(* IEC 61131-3 sources: MotionTestBenchMaster/Logical/00_AID/Libraries/Sidel_Libraries/Powertoys, 10 files *)

(* ---- Powertoys.typ ---- *)
(********************************************************************
 * COPYRIGHT -- Bernecker + Rainer
 ********************************************************************
 * Library: Powertoys
 * File: Powertoys.typ
 * Author: gibertinim
 * Created: March 27, 2014
 ********************************************************************
 * Data types of library Powertoys
 ********************************************************************)
(********************************                    CUSTOM LOGGER ENTRY                   ***********************************************************)

TYPE
	pwr_log_custom_entry : 	STRUCT  (*Custom logger entry string*)
		adr_string : UDINT; (*Address of the ascii string*)
		len : UDINT; (*Length of the binary memory data*)
		adr_mem : UDINT; (*Address to the binary memory data*)
		errorNum : UINT; (*Error number to write*)
		logLevel : USINT; (*Information level*)
	END_STRUCT;
END_TYPE

(*********************************                            HARDWARE LIST                          **************************************************************)

TYPE
	searchIO_info_typ : 	STRUCT  (*Hardware information list*)
		Path : STRING[80]; (*Station path*)
		ModelNumber : STRING[80]; (*Model number*)
		Name : STRING[80]; (*Hw name*)
		Serial : UDINT; (*Serial number*)
	END_STRUCT;
END_TYPE

(********************************                              AXIS INFORMATIONS                **************************************************************)

TYPE
	pwlInfo_typ : 	STRUCT  (*Powerlink node properties datatype*)
		number : USINT; (*Number of Powerlink Module*)
		path : STRING[80]; (*Path of Powerlink Module*)
		description : STRING[80]; (*Description of Powerlink Module*)
		name : STRING[80]; (*Name of Powerlink Module*)
		modelNumber : STRING[80]; (*Module number of powerlink *)
		present : BOOL; (*Enable blinking*)
	END_STRUCT;
END_TYPE

(* ---- CleanMgr.st ---- *)
(********************************************************************
 * COPYRIGHT --
 ********************************************************************
 * Library: Powertoys
 * File: CleanMgr.st
 * Author: Administrator
 * Created: January 09, 2015
 ********************************************************************
 * Implementation of library Powertoys
 ********************************************************************)

(* Clean old files from a folder *)
FUNCTION_BLOCK CleanMgr

	IF enable THEN
		(* Function block enabled *)
		CASE step OF

			0:
				busy 		:= TRUE;
				ready		:= FALSE;
				error 		:= FALSE;
				errorID 	:= ERR_FUB_BUSY;

				(* Getting the input parameters *)
				memset(ADR(dirInfoData), 0, SIZEOF(dirInfoData));
				memset(ADR(oldestFile), 0, SIZEOF(oldestFile));
				tRefresh.PT 		:= refreshTime;
				getDirInfo.pDevice	:= adrPath;
				getDirInfo.pPath	:= ADR('//');
				getLastFileName.pDevice := adrPath;
				getLastFileName.pPath := ADR('//');
				getLastFileName.option := fiFILE;
				getLastFileName.data_len := SIZEOF(dirInfoData);
				deleteFile.pDevice := adrPath;
				step := 1;

				IF (refreshTime <= T#10ms) OR (adrPath = 0) OR (nrElements = 0) THEN

					(* Refresh time too low, or path address = 0, or numer of elements invalid *)
					step 		:= 200;
					errorStep 	:= 0;
					error 		:= TRUE;
					errorID 	:= ERR_BUR_ILLPAR;

				END_IF;

			1:
				(* Waiting the refresh timer *)
				tRefresh.IN := TRUE;

				IF (adrPath <> getDirInfo.pDevice) THEN
					(* Incorrect path address *)
					step 		:= 200;
					errorStep 	:= 1;
					error 		:= TRUE;
					errorID 	:= ERR_BUR_ILLPAR;

				ELSIF tRefresh.Q THEN

					getDirInfo.enable := TRUE;
					IF (getDirInfo.status = ERR_FUB_BUSY) THEN
	 					step := 10;
					END_IF;

				END_IF;

			10:
				tRefresh.IN := FALSE;

				IF (adrPath <> getDirInfo.pDevice) THEN
					(* Incorrect path address *)
					step 		:= 200;
					errorStep 	:= 1;
					error 		:= TRUE;
					errorID 	:= ERR_BUR_ILLPAR;

				ELSIF (getDirInfo.status = ERR_OK) THEN
					fileFound := getDirInfo.filenum;
					step := 11;

				ELSIF (getDirInfo.status <> ERR_OK) AND (getDirInfo.status <> ERR_FUB_BUSY) THEN

					(* Error *)
					step 		:= 200;
					errorStep 	:= 10;
					error 		:= TRUE;
					errorID 	:= getDirInfo.status;
				END_IF;

			11:
				IF (getDirInfo.filenum > nrElements) THEN

					(* Proceeding with cleanup *)
					step := 20;
				ELSE
					step := 0;
				END_IF;
				getDirInfo.enable	:= FALSE;

			20:
				(* Clean up, finding the oldest file *)
				memset(ADR(dirInfoData), 0, SIZEOF(dirInfoData));
				memset(ADR(oldestFile), 0, SIZEOF(oldestFile));
				cnt := 0;
				getLastFileName.entry := cnt;
				getLastFileName.pData := ADR(oldestFile);
				IF (adrPath <> getLastFileName.pDevice) THEN
					(* Incorrect path address *)
					step 		:= 200;
					errorStep 	:= 20;
					error 		:= TRUE;
					errorID 	:= ERR_BUR_ILLPAR;
				ELSE
					getLastFileName.enable := TRUE;
					step := 21;
				END_IF

			21:
				IF (adrPath <> getLastFileName.pDevice) THEN
					(* Incorrect path address *)
					step 		:= 200;
					errorStep 	:= 21;
					error 		:= TRUE;
					errorID 	:= ERR_BUR_ILLPAR;

				ELSIF (getLastFileName.status = ERR_OK) THEN
					memset(ADR(dirInfoData), 0, SIZEOF(dirInfoData));
					getLastFileName.enable := FALSE;
					step := 22;

				ELSIF ((getLastFileName.status <> ERR_OK) AND (getLastFileName.status <> ERR_FUB_BUSY)) THEN
					(* Error *)
					step 		:= 200;
					errorStep 	:= 20;
					error 		:= TRUE;
					errorID 	:= getLastFileName.status;
				END_IF;

			22:

				getLastFileName.pData := ADR(dirInfoData);
				cnt := cnt + 1;
				getLastFileName.entry := cnt;

				IF (cnt < fileFound) THEN

					step := 23;

				ELSE
					(* search finished *)
					step := 30;
				END_IF;

			23:
				getLastFileName.enable := TRUE;
				IF (adrPath <> getLastFileName.pDevice) THEN
					(* Incorrect path address *)
					step 		:= 200;
					errorStep 	:= 23;
					error 		:= TRUE;
					errorID 	:= ERR_BUR_ILLPAR;

				ELSIF (getLastFileName.status = ERR_OK) THEN
					getLastFileName.enable := FALSE;
					step := 24;

				ELSIF ((getLastFileName.status <> ERR_OK) AND (getLastFileName.status <> ERR_FUB_BUSY) AND (getLastFileName.status <> ERR_FUB_ENABLE_FALSE)) THEN
					(* Error *)
					step 		:= 200;
					errorStep 	:= 22;
					error 		:= TRUE;
					errorID 	:= getLastFileName.status;
				END_IF;

			24:
				(* Checking the file timestamp *)
				IF (dirInfoData.Date < oldestFile.Date) THEN
					memcpy(ADR(oldestFile), ADR(dirInfoData), SIZEOF (oldestFile));

				END_IF;

				memset(ADR(dirInfoData),0,SIZEOF (dirInfoData));
				step := 22;

			30:
				(* Search finished, deleting the oldest file *)
				deleteFile.pName := ADR(oldestFile.Filename[0]);
				deleteFile.enable := TRUE;
				IF (adrPath <> deleteFile.pDevice) THEN
					(* Incorrect path address *)
					step 		:= 200;
					errorStep 	:= 30;
					error 		:= TRUE;
					errorID 	:= ERR_BUR_ILLPAR;
				ELSIF (deleteFile.status = ERR_OK) THEN
					deleteFile.enable := FALSE;
					IF (fileFound - 1 > nrElements) THEN
						getDirInfo.enable := TRUE;
						step := 10;
					ELSE
						step := 0;
					END_IF;

				ELSIF (deleteFile.status <> ERR_OK) AND (deleteFile.status <> ERR_FUB_ENABLE_FALSE) AND (deleteFile.status <> ERR_FUB_BUSY) THEN
					(* Error *)
					step 		:= 200;
					errorStep 	:= 30;
					error 		:= TRUE;
					errorID 	:= deleteFile.status;
				END_IF;

			200:
				(* Error state, resetting all the internal function block *)
				tRefresh.IN				:= FALSE;
				getDirInfo.enable		:= FALSE;
				getLastFileName.enable	:= FALSE;
				deleteFile.enable		:= FALSE;

		END_CASE;

	ELSE

		(* Function block disabled, resetting all the internal fubs *)
		busy 		:= FALSE;
		ready		:= FALSE;
		error 		:= TRUE;
		errorID 	:= ERR_FUB_ENABLE_FALSE;

		step 		:= 0;
		errorStep 	:= 0;
		cnt 		:= 0;
		tRefresh.IN				:= FALSE;
		getDirInfo.enable		:= FALSE;
		getLastFileName.enable	:= FALSE;
		deleteFile.enable		:= FALSE;
	END_IF;

	tRefresh();
	getDirInfo();
	getLastFileName();
	deleteFile();
END_FUNCTION_BLOCK

(* ---- CustomLogEntry.st ---- *)
(********************************************************************
 * COPYRIGHT -- Bernecker + Rainer
 ********************************************************************
 * Library: Powertoys
 * File: CustomLogEntry.st
 * Author: gibertinim
 * Created: March 27, 2014
 ********************************************************************
 * Implementation of library Powertoys
 ********************************************************************)

(* Write a custom entry into the specified logger *)
FUNCTION_BLOCK CustomLogEntry

	IF enable THEN

		pEntry ACCESS adrCustomEntry;

		CASE step OF

			0:	(*Check if Log exist*)
				LogInfo.Name	:= 'userlog';
				LogInfo.Execute	:= TRUE;
				errorID 		:= ERR_FUB_BUSY;
				busy			:= TRUE;
				error			:= FALSE;

				IF (LogInfo.StatusID = arEVENTLOG_ERR_LOGBOOK_NOT_FOUND) THEN
					step := 5;
					LogInfo.Execute	:= FALSE;
				ELSIF (LogInfo.Done AND LogInfo.StatusID = ERR_OK) THEN
					step 			:= 10;
					LogIdent		:= LogInfo.Ident;
					LogInfo.Execute	:= FALSE;
				END_IF

			5:	(*Create Log*)
				LogCreate.Name			:= 'userlog';
				LogCreate.Size			:= 4096;	//4096 BYTES
				LogCreate.Persistence	:= arEVENTLOG_PERSISTENCE_PERSIST;
				LogCreate.Execute		:= TRUE;
				errorID 				:= ERR_FUB_BUSY;
				busy					:= TRUE;
				error					:= FALSE;

				IF LogCreate.Error THEN
					step 		:= 200;
					error		:= TRUE;
					errorID		:= LogInfo.StatusID;
					errorStep	:= 1;
				ELSIF (LogCreate.Done AND LogInfo.StatusID = ERR_OK) THEN
					step				:= 10;
					LogIdent			:= LogCreate.Ident;
					LogCreate.Execute	:= FALSE;
				END_IF

			10:	(* Writing the logger informations  *)
				eventID := ArEventLogMakeEventID(
					Severity := pEntry.logLevel,
					Facility := 0,
					ErrorCode := pEntry.errorNum);

				LogWrite.EventID		:= eventID;
				LogWrite.Ident			:= LogIdent;
				LogWrite.AddData		:= pEntry.adr_string;
				LogWrite.AddDataSize	:= 80;
				LogWrite.AddDataFormat	:= 1;
				LogWrite.Execute		:= TRUE;

				(* Waiting until the log is written succesfully *)
				IF (LogWrite.Done AND LogWrite.StatusID = ERR_OK) THEN
					(* Log entry written succesfully*)
					step := 101;
					LogWrite.Execute := FALSE;
				ELSIF LogWrite.Error THEN
					(* Error occured while saving the logger *)
					errorStep	:= 10;
					errorID		:= LogWrite.StatusID;
					error		:= TRUE;
					step		:= 200;
				END_IF;

			101:
				done := TRUE;
				busy := FALSE;
				errorID := ERR_OK;

			200:
				(* Error step *)
				LogCreate.Execute	:= FALSE;
				LogWrite.Execute	:= FALSE;
				LogInfo.Execute		:= FALSE;
				done				:= TRUE;
				busy				:= FALSE;
		END_CASE;

	ELSE
		error				:= FALSE;
		errorID				:= ERR_FUB_ENABLE_FALSE;
		errorStep			:= 0;
		step	 			:= 0;
		LogCreate.Execute	:= FALSE;
		LogWrite.Execute	:= FALSE;
		LogInfo.Execute		:= FALSE;
		done				:= FALSE;
		busy				:= FALSE;

	END_IF;

	LogCreate();
	LogWrite();
	LogInfo();

END_FUNCTION_BLOCK

(* ---- PlkList.st ---- *)
(********************************************************************
 * COPYRIGHT --
 ********************************************************************
 * Library: Powertoys
 * File: Plk_list.st
 * Author: Administrator
 * Created: July 04, 2014
 ********************************************************************
 * Implementation of library Powertoys
 ********************************************************************)

(* Powerlink list *)
FUNCTION_BLOCK PlkList

	IF (enable	=	TRUE) THEN

		CASE step OF

			0: (* Choosing the operating mode
					0 = standard memory consumption
					1 = low memory consumption - slowest
				*)
				errorID 		:=	ERR_FUB_BUSY;
				busy			:=	TRUE;
				error			:=	FALSE;
				done			:= 	FALSE;

				IF (mode = 0) THEN
					step 		:= 1;
				ELSIF (mode = 1) THEN
					step 		:= 10;
				ELSE
					(* Wrong mode *)
					step		:= 200;
					error 		:= TRUE;
					errorID		:= ERR_NOTIMPLEMENTED;
					errorStep	:= 0;
					busy		:= FALSE;
					done		:= FALSE;
				END_IF;

			1:
				(* Getting the whole hardware list *)
				searchIO_0.adrSearchIO 	:= ADR(searchIoData);
				searchIO_0.mode 		:= asdiagALL;
				searchIO_0.wholeList	:= TRUE;
				searchIO_0.enable		:= TRUE;

				IF (searchIO_0.errorID = ERR_FUB_BUSY) THEN
					step := 2;
				END_IF;

			2:
				IF ((searchIO_0.errorID	=	ERR_OK) AND (searchIO_0.done = TRUE)) THEN

					(*resetting array and variables*)

					strcpy(ADR(tmpPlkInterface), ADR(plkInterface));
					strcat(ADR(tmpPlkInterface),ADR('.'));
					step		:=	3;
					indexInfo	:=	0;
					indexPwl	:=	0;

				ELSIF ((searchIO_0.errorID	<>	ERR_OK)	AND	(searchIO_0.errorID	<>	ERR_FUB_BUSY)) THEN

					(* Going to the error state *)
					errorID		:=	searchIO_0.errorID;
					errorStep	:=	1;
					step		:=	200;
					error		:=	TRUE;
				END_IF

			3: (*saving inside an array	(ArrayStringTemp) the path hardware longer than plk inteface*)
			IF (indexInfo	<	searchIO_0.nrEntries)	THEN

				(* Ci metto tutto quello dopo SS1.IF1
					Es:
					ST2
					ST3
					ST5.IF1

				*)
				IF 	strlen(ADR(searchIoData[indexInfo].Path))	>=	strlen(ADR(tmpPlkInterface))	THEN
					strcpy(ADR(ArrayStringTemp[indexPwl]),(ADR(searchIoData[indexInfo].Path)+ strlen(ADR(tmpPlkInterface))));
					arrayIndexPwl[indexPwl]	:=	indexInfo;
					indexPwl				:=	indexPwl+1;
				END_IF;

				indexInfo	:=	indexInfo+1;
			ELSE
				step		:=	4;
				oldIndexPwl :=	indexPwl;

				indexPwl	:=	0;

				indexInfo	:=	0;
				indexPwl2	:=	0;
				dotFound	:=	FALSE;

				END_IF;

		4:
			(*Finding dot or string null inside elements of temp array*)
			IF (indexPwl	<	strlen(ADR(ArrayStringTemp[indexInfo]))	OR	strlen(ADR(ArrayStringTemp[indexInfo]))	=	0 )	THEN

				IF (memcmp(ADR(ArrayStringTemp[indexInfo])+indexPwl,ADR('.'),1)	=0	)	THEN
					step		:=	5;
					indexPwl	:=	0;
					dotFound 	:= TRUE;
				END_IF;

			ELSE
				step		:=	5;
				indexPwl	:=	0;

			END_IF;
			indexPwl	:=	indexPwl+1;

		5:

			(*if there isn't a dot, the string is our node powerlink*)
			IF (dotFound	=	FALSE) THEN

				pData ACCESS (adrPlkInfo + indexPwl2*SIZEOF(pData));
				pData.number	:=	arrayIndexPwl[indexInfo];

				IF strlen(ADR(searchIoData[arrayIndexPwl[indexInfo]].ModelNumber))	<>	0 	AND
					pData.number	<>	0									THEN
					(* Powerlink node present *)
					pData.present	:=	TRUE;
				ELSE
					(* Powerlink node not present *)
					pData.present	:=	FALSE;
				END_IF;

				(*Copying information about powerlink node*)
				strcpy(ADR(pData.path),						ADR(ArrayStringTemp[indexInfo]));
				strcpy(ADR(pData.modelNumber),				ADR(searchIoData[arrayIndexPwl[indexInfo]].ModelNumber));
				strcpy(ADR(pData.name),						ADR(searchIoData[arrayIndexPwl[indexInfo]].Name));
				strcpy(ADR(ArrayStringTemp2[indexPwl2]),	ADR(ArrayStringTemp[indexInfo]));
				arrayIndexPwl2[indexPwl2]					:=	arrayIndexPwl[indexInfo];
				indexPwl2									:=	indexPwl2+1;

			END_IF;
			(**)
			indexInfo	:=	indexInfo+1;
			IF (indexInfo	<	oldIndexPwl) THEN

				dotFound	:=	FALSE;
				step	:=	4;

			ELSE

				step	:=	6;

			END_IF;

		6:
			busy := FALSE;
			done := TRUE;
			errorID := ERR_OK;

			entryFound := indexPwl2;

			10:
				(* Low memory consumption mode *)
				(* In this mode each entry is processe one by one instead of processing the whole list *)
				(* Getting the whole hardware list *)
				searchIO_0.adrSearchIO 	:= ADR(searchIoData);
				searchIO_0.mode 		:= asdiagALL;
				searchIO_0.wholeList	:= FALSE;
				searchIO_0.enable		:= TRUE;
				indexInfo 				:= 0;
				indexPwl2 				:= 0;
				(* Getting informations from the first hw found *)
				searchIO_0.stationIndex	:= 0;

				IF (searchIO_0.errorID = ERR_FUB_BUSY) THEN
					step := 11;
				END_IF;

			11:

				IF ((searchIO_0.errorID	=	ERR_OK) AND (searchIO_0.done = TRUE)) THEN

					(*resetting array and variables*)

					strcpy(ADR(tmpPlkInterface), ADR(plkInterface));
					strcat(ADR(tmpPlkInterface),ADR('.'));
					step		:=	12;
					nrIO 		:= searchIO_0.nrEntries;

				ELSIF ((searchIO_0.errorID	<>	ERR_OK)	AND	(searchIO_0.errorID	<>	ERR_FUB_BUSY)) THEN
					(* Going to the error state *)
					errorID		:=	searchIO_0.errorID;
					errorStep	:=	10;
					step		:=	200;
					error		:=	TRUE;
				END_IF

			12:
				 (* Se la lunghezza del path trovato dalla search io è maggiore o uguale a quello dell'interfaccia powerlink, allora è un probabile nodo powerlink *)
				(* Copio nella variabile temporanea solo quello che viene dopo i caratteri che compongono l'interfaccia powerlink:
				Es: Ci metto tutto quello dopo SS1.IF1

				in powerlink if ci deve finire 'SS1.IF1.'

				Se per esempio avremo come entry:
				SS1.IF1
				SS1.IF1.ST2
				SS1.IF1.ST3
				SSI.IF1.ST5.IF8

				RIMARRANNO

				ST2
				ST3
				ST5.IF8

				*)
				IF 	strlen(ADR(searchIoData[0].Path))	>=	strlen(ADR(tmpPlkInterface))	THEN

					(* Possible powerlink node *)
					strcpy(ADR(ArrayStringTemp[0]),(ADR(searchIoData[0].Path)+ strlen(ADR(tmpPlkInterface))));

					arrayIndexPwl[0]	:=	indexInfo;

					step := 13;

				ELSE
					(* Not a powerlink node *)
					step := 100;
				END_IF;

			13:
				(* If the remaining temporary string is empty, this is the powerlink inferface, not the powerlink node  *)

				IF (strlen(ADR(ArrayStringTemp[0])) <> 0) THEN

					(* Possible powerlink node *)
					tmpCnt		:= 0;
					step		:= 14;
				ELSE
					(* Not a powerlink node *)
					step		:= 100;
				END_IF;

			14:
				(* I have only something like:
				ST5
				ST41
				ST123
				ST41.IFblablabla
				ST12

				I can say that if there is not the dot, this is a powerlink node

				SEARCHING inside of the string if there is the dot
				*)
				IF (tmpCnt < strlen(ADR(ArrayStringTemp[0]))) THEN

					IF (memcmp(ADR(ArrayStringTemp[0])+tmpCnt,ADR('.'),1)	= 0	) THEN

						(* Dot found, this is not a powerlink node *)
						step := 100;

					ELSE
						tmpCnt := tmpCnt + 1;
					END_IF;

				ELSE
					(* This is a powerlink node *)
					step := 15;
				END_IF;

			15:
				(* Collecting data of the powerlink node *)
				pData ACCESS (adrPlkInfo + indexPwl2*SIZEOF(pData));
				pData.number	:=	indexInfo;

				IF strlen(ADR(searchIoData[0].ModelNumber))	<>	0 	AND
					pData.number	<>	0									THEN
					(* Powerlink node present *)
					pData.present	:=	TRUE;
				ELSE
					(* Powerlink node not present *)
					pData.present	:=	FALSE;
				END_IF;

				(*Copying information about powerlink node*)
				strcpy(ADR(pData.path),						ADR(ArrayStringTemp[0]));
				strcpy(ADR(pData.modelNumber),				ADR(searchIoData[0].ModelNumber));
				strcpy(ADR(pData.name),						ADR(searchIoData[0].Name));
				indexPwl2									:=	indexPwl2+1;

				step	:=	100;

			100:
				(* Not a powerlink node, processing a new entry *)
				searchIO_0.enable		:= FALSE;

				IF (searchIO_0.errorID = ERR_FUB_ENABLE_FALSE) THEN
					indexInfo := indexInfo + 1;
					step := 101;
				END_IF;

			101:
				(* Checking if I have to read an other entry *)
				IF ((indexInfo < nrIO)AND(indexPwl < nrEntry))  THEN

					(* Cleaning temporary variables *)
					memset(ADR(searchIoData),0,SIZEOF(searchIoData));

					(* Going to process a new entry *)
					step := 102;

				ELSE

					(* Sequence finished *)
					step := 120;

				END_IF;

			102:
				(* Reading a new search IO entry *)
				searchIO_0.adrSearchIO 	:= ADR(searchIoData);
				searchIO_0.mode 		:= asdiagALL;
				searchIO_0.wholeList	:= FALSE;
				searchIO_0.enable		:= TRUE;

				(* Getting informations from the first hw found *)
				searchIO_0.stationIndex	:= indexInfo;

				IF (searchIO_0.errorID = ERR_FUB_BUSY) THEN
					step := 103;
				END_IF;

			103:

				IF ((searchIO_0.errorID	=	ERR_OK) AND (searchIO_0.done = TRUE)) THEN

					(*resetting array and variables*)

					step		:=	12;
					nrIO 		:= searchIO_0.nrEntries;

				ELSIF ((searchIO_0.errorID	<>	ERR_OK)	AND	(searchIO_0.errorID	<>	ERR_FUB_BUSY)) THEN
					(* Going to the error state *)
					errorID		:=	searchIO_0.errorID;
					errorStep	:=	102;
					step		:=	200;
					error		:=	TRUE;
				END_IF

			120:
			(* Sequence completed *)
				done 				:= TRUE;
				busy 				:= FALSE;
				error 				:= FALSE;
				errorID				:= ERR_OK;
				searchIO_0.enable	:= FALSE;
				entryFound := indexPwl2;

			200:
				(* Error state, disabling all the used function block and waiting  for enable = false *)
				searchIO_0.enable 	:= FALSE;

		END_CASE;

	ELSE
		(* Function block not enabled *)
		error				:= TRUE;
		errorID				:= ERR_FUB_ENABLE_FALSE;

		(* Resetting  the internal variables *)
		errorStep			:= 0;
		step	 			:= 0;

		memset(ADR(arrayIndexPwl),		0,	SIZEOF(arrayIndexPwl));
		memset(ADR(ArrayStringTemp),	0,	SIZEOF(ArrayStringTemp));
		memset(ADR(arrayIndexPwl2),		0,	SIZEOF(arrayIndexPwl2));
		memset(ADR(ArrayStringTemp2),	0,	SIZEOF(ArrayStringTemp2));
		memset(ADR(tmpPlkInterface),	0,	SIZEOF(tmpPlkInterface));

		step		:=	0;
		indexInfo	:=	0;
		indexPwl	:=	0;
		indexPwl2	:=	0;
		entryFound 	:= 	0;
		nrIO		:=	0;
		done				:= FALSE;
		busy				:= FALSE;

		(* Disabling the block *)
		searchIO_0.enable 	:= FALSE;

	END_IF;

	(*Function Block Call*)
	searchIO_0();
END_FUNCTION_BLOCK

(* ---- Powertoys.fun ---- *)
(********************************************************************
 * COPYRIGHT -- Bernecker + Rainer
 ********************************************************************
 * Library: Powertoys
 * File: Powertoys.fun
 * Author: gibertinim
 * Created: March 27, 2014
 ********************************************************************
 * Functions and function blocks of library Powertoys
 ********************************************************************)

FUNCTION_BLOCK CustomLogEntry (*Write a custom entry into the specified logger*)
	VAR_INPUT
		enable : BOOL; (*Enable the function block*)
		adrCustomEntry : UDINT; (*Address of the custom entry*)
	END_VAR
	VAR_OUTPUT
		busy : BOOL; (*True when the function block is busy*)
		error : BOOL; (*True when the function block is in error*)
		errorID : DINT; (*Current error ID*)
		done : BOOL; (*True when the entry is succesfully written*)
	END_VAR
	VAR
		LogCreate : ArEventLogCreate;
		LogInfo : ArEventLogGetIdent; (*Get the information from the specified logger*)
		LogWrite : ArEventLogWrite; (*Write the entry into the logger*)
		eventID : DINT;
		errorStep : UINT; (*Internal error step*)
		pEntry : REFERENCE TO pwr_log_custom_entry; (*Pointer to the custom entry*)
		step : USINT; (*Internal fub step*)
		LogIdent : ArEventLogIdentType;
	END_VAR
END_FUNCTION_BLOCK

FUNCTION_BLOCK SearchIO (*Function Block to show hardware list component*)
	VAR_INPUT
		enable : BOOL; (*Enable the function block*)
		adrSearchIO : UDINT; (*Address of the search io data structure*)
		wholeList : BOOL; (*True to create the hw list, false for a single entries*)
		stationIndex : UDINT; (*Station index number (used only if wholeList = FALSE)*)
		mode : UDINT; (*Operating mode*)
	END_VAR
	VAR_OUTPUT
		busy : BOOL; (*True when the function block is busy*)
		done : BOOL; (*True when the data are ready*)
		error : BOOL; (*True when the function block is in error*)
		errorID : UINT; (*Current error ID*)
		nrEntries : UDINT; (*Number of entries found*)
	END_VAR
	VAR
		counter : UDINT; (*Internal counter*)
		ident : UDINT; (*Identifier*)
		FB_DiagGetStrInfo : DiagGetStrInfo; (*Get the string information of the module*)
		FB_DiagCreateInfo : DiagCreateInfo; (*Collect the information of the specified module*)
		FB_DiagGetNumInfo : DiagGetNumInfo; (*Get the numeric information from the specified module*)
		step : USINT; (*Internal fub step*)
		errorStep : USINT; (*Internal error step*)
		pData : REFERENCE TO searchIO_info_typ; (*Pointer to the data structure*)
	END_VAR
END_FUNCTION_BLOCK

FUNCTION_BLOCK PlkList (*Powerlink list*)
	VAR_INPUT
		enable : BOOL; (*Enable the function block*)
		adrPlkInfo : UDINT; (*Address of the powerlink information list*)
		mode : USINT; (*Fub operating mode (0 high memory usage, 1 low memory usage)*)
		nrEntry : UDINT; (*Number of powerlink elements to write on the list*)
		plkInterface : STRING[80]; (*String initialize a lenght of powerlink path*)
	END_VAR
	VAR_OUTPUT
		done : BOOL; (*Powerlink list complete*)
		busy : BOOL; (*Function block busy*)
		error : BOOL; (*Function block in error*)
		errorID : UINT; (*Function block error ID*)
		entryFound : USINT; (*Number of powerlink node in the configuration*)
	END_VAR
	VAR
		errorStep : USINT; (*Internal error step*)
		step : USINT; (*Internal step*)
		pData : REFERENCE TO pwlInfo_typ; (*Pointer to the powerlink list*)
		searchIO_0 : SearchIO; (*Search IO informations*)
		searchIoData : ARRAY[0..253] OF searchIO_info_typ; (*Search IO informations strusture*)
		arrayIndexPwl : ARRAY[0..253] OF USINT; (*Array to save index of hardware list complete*)
		arrayIndexPwl2 : ARRAY[0..253] OF USINT; (*Array to save index when dot is not finding*)
		ArrayStringTemp : ARRAY[0..253] OF STRING[80]; (*Array temp for saving name of powerlink node longer than plkinterface*)
		ArrayStringTemp2 : ARRAY[0..253] OF STRING[80]; (*Array to save path name when dot is not finding*)
		indexInfo : USINT; (*Index of number entries of harware list complete*)
		tmpPlkInterface : STRING[80]; (*Internal powerlink interface name*)
		indexPwl : USINT; (*Index of array for saving name of powerlink node longer than plkinterface*)
		oldIndexPwl : USINT; (*savind old index powerlink*)
		indexPwl2 : USINT; (*Index of array when dot is not finding*)
		dotFound : BOOL; (*Finding dot inside an array*)
		nrIO : UDINT; (*Number of IO found with the SEARCH IO fub*)
		tmpCnt : USINT; (*Temporary counter*)
	END_VAR
END_FUNCTION_BLOCK

FUNCTION_BLOCK profiMan (*Profiler archive manager*)
	VAR_INPUT
		enable : BOOL; (*Enable the function block*)
		refreshTime : TIME; (*Automatic refresh time*)
		maxArchive : USINT; (*Maximum number of profiler acrhive stored*)
		archiveListADR : UDINT; (*Address of the archive list*)
	END_VAR
	VAR_OUTPUT
		errorID : UINT; (*Current error ID*)
		valid : BOOL; (*True when the output data are valid*)
		error : BOOL; (*True when the function block is in error*)
		profilerStatus : USINT; (*Profiler status*)
		archiveFound : UDINT; (*Number of profiler archive found*)
		busy : BOOL; (*True when the function block is busy*)
		profStateActive : BOOL; (*Profiler active. AR profiler is ready.*)
		profStateStopped : BOOL; (*Data recording stopped.*)
		profStateRunning : BOOL; (*Data being recorded.*)
		profStateReady : BOOL; (*Data recording completed. The data module is ready to be evaluated (AS profiler).*)
		profStateR2R : BOOL; (*Ready to start. A profiling definition was installed successfully and can be started.*)
		profStateInactive : BOOL; (*Profiler inactive. Profiling cannot be carried out (AR profiler disabled in Sysconf).*)
		profStateR2Rman : BOOL; (*Ready to start (startup install). The profiler definition was installed successfully with the profMODE_NOAUTOSTART mode and can be started.*)
	END_VAR
	VAR
		pArchiveList : REFERENCE TO PROFILER_MODINFO; (*Pointer to the archive list*)
		step : USINT; (*Internal state machine step*)
		getProfStatus : LogStateGet; (*Get the status of the profiler*)
		errorStep : USINT; (*Internal error step*)
		getProfArchInfo : LogArchInfo; (*Gets profiler's archive informations*)
		refresh : TON; (*Refresh timer*)
	END_VAR
END_FUNCTION_BLOCK

FUNCTION_BLOCK sdmMAN (*Sdm configuration manager*)
	VAR_INPUT
		enable : BOOL; (*Enable the function block*)
		mode : USINT; (*Function block operating mode: 0 - SDM on, 1 - SDM off, 2 SDM status manual*)
		reqSDMstatus : UDINT; (*Requested SDM status*)
		pDumpDevice : UDINT; (*Pointer to the file device of the system dump*)
	END_VAR
	VAR_OUTPUT
		sdmStatus : UDINT; (*Actual SDM status*)
		busy : BOOL; (*True when the function block is working*)
		ready : BOOL; (*True when the function block is waiting for a change of reqSDMstatus*)
		error : BOOL; (*True when the function block is in error*)
		errorID : UINT; (*Actual error ID*)
		internalError : BOOL; (*Internal error*)
		errorStep : USINT; (*Actual error step*)
	END_VAR
	VAR
		old_mode : USINT; (*Old mode*)
		setSDMstatus : CfgSetSdmStatus; (*Set the sdm status*)
		getSDMstatus : CfgGetSdmStatus; (*Get the sdm status*)
		oldSdmStatus : UDINT; (*Old SDM status*)
		step : USINT; (*Internal function block step*)
		writeLogFlag : BOOL; (*Write an entry into the logger*)
		errorStepString : STRING[80]; (*Error step as string*)
		errorString : STRING[80]; (*Error string*)
		errorEntry : pwr_log_custom_entry; (*Log entry*)
		sDump : SdmSystemDump; (*Makes the system dump*)
		writeError : CustomLogEntry; (*Write the error into the user logger*)
	END_VAR
END_FUNCTION_BLOCK

FUNCTION_BLOCK CleanMgr (*Clean old files from a folder*)
	VAR_INPUT
		enable : BOOL; (*Enable the function block*)
		refreshTime : TIME; (*Folder refresh time*)
		adrPath : UDINT; (*Address of the path to clean*)
		nrElements : UDINT; (*Number of elements to keep into the folder*)
	END_VAR
	VAR_OUTPUT
		busy : BOOL; (*True when then the function block is busy*)
		ready : BOOL; (*True when the function block is ready*)
		error : BOOL; (*True when the function block is in error*)
		errorID : UINT; (*Function block error ID*)
	END_VAR
	VAR
		cnt : UDINT; (*Internal counter*)
		oldestFile : fiDIR_READ_DATA; (*Oldest filename*)
		fileFound : UDINT; (*Number of file found*)
		dirInfoData : fiDIR_READ_DATA; (*Information red*)
		step : USINT; (*Internal step*)
		errorStep : USINT; (*Internal error step*)
		tRefresh : TON; (*Refresh timer*)
		getLastFileName : DirRead; (*Get the last filename*)
		deleteFile : FileDelete; (*Delete one file*)
		getDirInfo : DirInfo; (*Get the directory informations*)
	END_VAR
END_FUNCTION_BLOCK

FUNCTION_BLOCK saveNCT (*Save the network comand trace into one file*)
	VAR_INPUT
		enable : BOOL; (*Enable the function block*)
		fName : STRING[32]; (*Output filename*)
		mode : USINT; (*0 - Filename only, 1 - Filename with timestamp*)
		deviceName : STRING[32]; (*Device name*)
	END_VAR
	VAR_OUTPUT
		busy : BOOL; (*True when the function block is busy*)
		done : BOOL; (*True when the function block has finished to work*)
		error : BOOL; (*True when the function block is in error*)
		traceError : MC_ERRORRECORD_REF; (*Trace recorded error*)
		errorStep : USINT; (*Error Step*)
		errorID : UINT; (*Actual error ID*)
	END_VAR
	VAR
		NetTraceConfig : MC_NETTRACECONFIG_REF; (*Network command trace upload config*)
		NetTraceStatusConfig : MC_NETTRACECONFIG_REF; (*Network command trace status configuration*)
		MC_BR_ReadNetTraceStatus_0 : MC_BR_ReadNetTraceStatus; (*Network command trace status*)
		MC_BR_NetTrace_0 : MC_BR_NetTrace; (*Network command trace management fub*)
		step : USINT; (*Internal step*)
	END_VAR
END_FUNCTION_BLOCK

(* ---- profiMan.st ---- *)
(********************************************************************
 * COPYRIGHT --
 ********************************************************************
 * Library: Powertoys
 * File: profiMan.st
 * Author: Administrator
 * Created: July 24, 2014
 ********************************************************************
 * Implementation of library Powertoys
 ********************************************************************)

(* Profiler archive manager *)

FUNCTION_BLOCK profiMan

	IF enable THEN

		CASE step OF

			(* GETTING THE PROFILER STATUS *)
			0:
				refresh.IN := FALSE;
				IF (getProfStatus.status = ERR_FUB_ENABLE_FALSE) THEN
					step := 1;
				END_IF;

			1:
				getProfStatus.enable := TRUE;

				IF (getProfStatus.status = ERR_OK) THEN
					step := 2;
					profilerStatus := getProfStatus.logstate;

				ELSIF (getProfStatus.status <> ERR_OK) AND (getProfStatus.status <> ERR_FUB_BUSY) AND (getProfStatus.status <> ERR_FUB_ENABLE_FALSE) THEN

					(* An error occured *)
					step		:= 200;
					errorStep	:= 1;
					error 		:= TRUE;
					errorID		:= getProfStatus.status;
				END_IF;

			2:
				profStateInactive	:= FALSE;
				profStateActive		:= FALSE;
				profStateStopped	:= FALSE;
				profStateRunning	:= FALSE;
				profStateReady		:= FALSE;
				profStateR2R		:= FALSE;
				profStateR2Rman		:= FALSE;

				CASE profilerStatus OF

					profSTATE_INACTIVE:
						(* Profiler inactive. Profiling cannot be carried out (AR profiler disabled in Sysconf). *)
						profStateInactive	:= TRUE;

					profSTATE_ACTIVE:
						(* Profiler active. AR profiler is ready. *)
						profStateActive		:= TRUE;

					profSTATE_STOPPED:
						(* Data recording stopped. *)
						profStateStopped	:= TRUE;

					profSTATE_RUNNING:
						(* Data being recorded. *)
						profStateRunning	:= TRUE;

					profSTATE_READY:
						(* Data recording completed. The data module is ready to be evaluated (AS profiler). *)
						profStateReady		:= TRUE;

					profSTATE_R2R:
						(* Ready to start. A profiling definition was installed successfully and can be started. *)
						profStateR2R		:= TRUE;

					profSTATE_R2R_MAN:
						(* Ready to start (startup install). The profiler definition was installed successfully with the profMODE_NOAUTOSTART mode and can be started. *)
						profStateR2Rman		:= TRUE;

				END_CASE;

				getProfStatus.enable := FALSE;

				IF (getProfStatus.status = ERR_FUB_ENABLE_FALSE) AND (getProfArchInfo.status = ERR_FUB_ENABLE_FALSE) THEN
					step := 3;
				END_IF;

			3:
				(* Checking that the archivwe list address is different than 0 *)
				IF (archiveListADR <> 0) AND (refreshTime <> 0) THEN

					(* There is a memory address *)
					step := 4;

				ELSE

					(* Address invalid *)
					errorStep	:= 3;
					step 		:= 200;
					error		:= TRUE;
					busy		:= FALSE;
					valid		:= FALSE;
					errorID		:= ERR_NOTIMPLEMENTED;

				END_IF;

		4:		(* List te number of profiler archives *)
				getProfArchInfo.enable		:= TRUE;
				getProfArchInfo.pInfo		:= archiveListADR;
				getProfArchInfo.maxEntries	:= maxArchive;

				IF (getProfArchInfo.status = ERR_FUB_BUSY) THEN
					step := 5;
				ELSIF (getProfArchInfo.status <> ERR_OK) AND (getProfArchInfo.status <> ERR_FUB_BUSY) AND (getProfArchInfo.status <> ERR_FUB_ENABLE_FALSE) THEN
					step 		:= 200;
					errorStep	:= 4;
					error 		:= TRUE;
					errorID 	:= getProfArchInfo.status;
					busy 		:= FALSE;
					valid		:= FALSE;

				END_IF;

			5:
				IF (getProfArchInfo.status = ERR_OK) THEN
					step := 6;
					archiveFound := getProfArchInfo.entries;

				ELSIF (getProfArchInfo.status <> ERR_OK) AND (getProfArchInfo.status <> ERR_FUB_BUSY) AND (getProfArchInfo.status <> ERR_FUB_ENABLE_FALSE) THEN
					step 		:= 200;
					errorStep	:= 5;
					error 		:= TRUE;
					errorID 	:= getProfArchInfo.status;
					busy 		:= FALSE;
					valid		:= FALSE;
				END_IF;

			6:

				getProfArchInfo.enable	:= FALSE;

				(* Checking if I have to delete some old profiler archive *)
				refresh.IN := TRUE;
				refresh.PT := refreshTime;

				IF (refresh.Q = TRUE) THEN
					step := 0;

				END_IF;

			200:
				getProfStatus.enable 	:= FALSE;
				refresh.IN 				:= FALSE;
				getProfArchInfo.enable	:= FALSE;

		END_CASE;

	ELSE

		busy			:= FALSE;
		error			:= TRUE;
		errorID			:= ERR_FUB_ENABLE_FALSE;
		valid			:= FALSE;
		profilerStatus	:= 254;

		step 			:= 0;
		errorStep		:= 0;
		archiveFound	:= 0;

		profStateInactive	:= FALSE;
		profStateActive		:= FALSE;
		profStateStopped	:= FALSE;
		profStateRunning	:= FALSE;
		profStateReady		:= FALSE;
		profStateR2R		:= FALSE;
		profStateR2Rman		:= FALSE;

		(* Disabling alla the used FUNCTION blocks *)
		refresh.IN				:= FALSE;
		getProfStatus.enable	:= FALSE;

		getProfArchInfo.enable	:= FALSE;

	END_IF;

	getProfStatus();
	refresh();
	getProfArchInfo();

END_FUNCTION_BLOCK

(* ---- saveNCT.st ---- *)
(********************************************************************
 * COPYRIGHT --
 ********************************************************************
 * Library: Powertoys
 * File: saveNCT.st
 * Author: Massimo Gibertini - B&R
 * Created: January 20, 2015
 ********************************************************************
 * Implementation of library Powertoys
 ********************************************************************)

(* Save the network comand trace into one file *)
FUNCTION_BLOCK saveNCT

	IF enable THEN
		CASE step OF
			0:
				error 		:= FALSE;
				busy		:= TRUE;
				done		:= FALSE;
				errorID 	:= ERR_FUB_BUSY;

				IF (strlen(ADR(fName)) <> 0) AND (strlen(ADR(deviceName)) <> 0) THEN
					NetTraceStatusConfig.NetTrace.Type			:= mcNET_TRACE_GLOBAL;
					NetTraceConfig.NetTrace.Type				:= mcNET_TRACE_GLOBAL;
					NetTraceConfig.DatObj.Name					:= fName;

					CASE mode OF
						0:
							NetTraceConfig.DatObj.Type					:= mcFILE;

						1:
							NetTraceConfig.DatObj.Type					:= mcFILE + mcADD_DATE_TIME;

					END_CASE;

					NetTraceConfig.DatObj.Format				:= 0;
					NetTraceConfig.DatObj.Device				:= deviceName;
					MC_BR_NetTrace_0.Configuration				:= NetTraceConfig;
					MC_BR_NetTrace_0.Command					:= mcSAVE;
					MC_BR_ReadNetTraceStatus_0.Configuration	:= NetTraceStatusConfig;
					MC_BR_ReadNetTraceStatus_0.Enable			:= TRUE;

					IF MC_BR_ReadNetTraceStatus_0.Busy THEN
						step := 1;
					END_IF;
				ELSE
					error 		:= TRUE;
					errorID		:= ERR_BUR_ILLPAR;
					errorStep	:= 0;
					step		:= 200;
				END_IF;

			1:
				IF (MC_BR_ReadNetTraceStatus_0.Valid AND MC_BR_ReadNetTraceStatus_0.TraceState = mcOFF) THEN
					(* Data not written to the network command trace *)
					step := 10;
				ELSIF (MC_BR_ReadNetTraceStatus_0.Valid AND MC_BR_ReadNetTraceStatus_0.TraceState = mcON) THEN
					(* Data written to the network command trace *)
					step := 20;
				ELSIF (MC_BR_ReadNetTraceStatus_0.Error) THEN
					error		:= TRUE;
					errorStep	:= 1;
					errorID		:= MC_BR_ReadNetTraceStatus_0.ErrorID;
					step 		:= 200;
				END_IF;

			10:
				(* Network command trace data not available *)
				MC_BR_ReadNetTraceStatus_0.Enable	:= FALSE;
				error 		:= TRUE;
				busy		:= FALSE;
				done		:= TRUE;
				errorID 	:= ERR_OK;

			20:
				(* Network command trace data available *)
				MC_BR_ReadNetTraceStatus_0.Enable	:= FALSE;
				MC_BR_NetTrace_0.Execute 			:= TRUE;
				IF MC_BR_NetTrace_0.Busy THEN
					step := 21;
				END_IF;

			21:
				IF MC_BR_NetTrace_0.Done THEN
					step := 30;
				ELSIF MC_BR_NetTrace_0.Error THEN
					traceError 	:= MC_BR_NetTrace_0.ErrorRecord;
					errorID 	:= MC_BR_NetTrace_0.ErrorID;
					error 		:= TRUE;
					errorStep 	:= 21;
					step 		:= 200;
				END_IF;
			30:
				(* NCT Saved *)
				MC_BR_NetTrace_0.Execute			:= FALSE;

				error 		:= FALSE;
				busy		:= FALSE;
				done		:= TRUE;
				errorID 	:= ERR_OK;

			200:
				(* ERROR *)
				MC_BR_NetTrace_0.Execute			:= FALSE;
				MC_BR_ReadNetTraceStatus_0.Enable	:= FALSE;

		END_CASE;

	ELSE

		MC_BR_NetTrace_0.Execute			:= FALSE;
		MC_BR_ReadNetTraceStatus_0.Enable	:= FALSE;
		step 		:= 0;

		error 		:= TRUE;
		busy		:= FALSE;
		done		:= FALSE;
		errorStep	:= 0;
		errorID 	:= ERR_FUB_ENABLE_FALSE;

	END_IF;

	MC_BR_NetTrace_0();
	MC_BR_ReadNetTraceStatus_0();

END_FUNCTION_BLOCK

(* ---- sdmMAN.st ---- *)
(********************************************************************
 * COPYRIGHT --
 ********************************************************************
 * Library: Powertoys
 * File: sdmMAN.st
 * Author: Administrator
 * Created: December 18, 2014
 ********************************************************************
 * Implementation of library Powertoys
 ********************************************************************)

(* TODO: Add your comment here *)
FUNCTION_BLOCK sdmMAN

	IF enable THEN

		CASE step OF

			0:
				busy		:= TRUE;
				ready		:= FALSE;
				error		:= FALSE;
				errorID		:= ERR_FUB_BUSY;

				(* Getting the required operating mode *)
				old_mode	:= mode;

				IF old_mode <= 3 THEN
					CASE old_mode OF
						0:
							(* If SDM is off then switch it on *)
							step 		:= 10;
						1:
							(* If SDM is on the switch it off *)
							step 		:= 20;
						2:
							(* Manual handling of the sdm configuration *)
							step 		:= 30;

						3:
							(* SYSTEM DUMP 	*)
							step		:= 40;

					END_CASE;

				ELSE
					error		:= TRUE;
					errorID		:= ERR_NOTIMPLEMENTED;
					errorStep	:= 0;
					step 		:= 200;
				END_IF;

			10:
				(* If SDM is off then switch it on *)
				IF (old_mode <> mode) THEN
					(* Operating mode shanged, returning at the beginning *)
					step				:= 0;
				ELSIF (getSDMstatus.enable = FALSE) AND (getSDMstatus.status = ERR_FUB_ENABLE_FALSE) THEN
					getSDMstatus.enable := TRUE;
					step				:= 11;
				END_IF;

			11:
				IF (old_mode <> mode) THEN
					(* Operating mode shanged, returning at the beginning *)
					step			:= 100;
				ELSIF (getSDMstatus.status = ERR_OK) AND (getSDMstatus.run = cfgSTATUS_SDM_ENABLED) THEN
					sdmStatus 		:= CST_SDM_ACTIVE;
					step			:= 18;
				ELSIF (getSDMstatus.status = ERR_OK) AND (getSDMstatus.run = cfgSTATUS_SDM_DISABLED) THEN
					sdmStatus 		:= CST_SDM_DISABLE;
					step			:= 12;
					writeLogFlag 	:= TRUE;
				ELSIF (getSDMstatus.status <> ERR_OK) AND (getSDMstatus.status <> ERR_FUB_BUSY) THEN
					(* Error occured *)
					error			:= TRUE;
					errorID			:= getSDMstatus.status;
					errorStep		:= 10;
					step 			:= 200;
				END_IF;

			12:
				(* Activating the SDM *)
				getSDMstatus.enable		:= FALSE;
				setSDMstatus.enable		:= FALSE;

				IF (old_mode <> mode) THEN
					(* Operating mode shanged, returning at the beginning *)
					step				:= 100;
				ELSIF (getSDMstatus.status = ERR_FUB_ENABLE_FALSE) AND (setSDMstatus.status = ERR_FUB_ENABLE_FALSE) THEN
					setSDMstatus.enable	:= TRUE;
					setSDMstatus.start	:= cfgOPTION_ENABLE_SDM;
					step				:= 13;
				END_IF;

			13:
				IF (old_mode <> mode) THEN
					(* Operating mode shanged, returning at the beginning *)
					step		:= 100;
				ELSIF (setSDMstatus.status = ERR_OK) THEN
					step		:= 14;
				ELSIF (setSDMstatus.status <> ERR_OK) AND (setSDMstatus.status <> ERR_FUB_BUSY) THEN
					(* Error occured *)
					error		:= TRUE;
					errorID		:= setSDMstatus.status;
					errorStep	:= 12;
					step 		:= 200;
				END_IF;

			14:
				(* Reading the sdm status *)
				setSDMstatus.enable		:= FALSE;

				IF (old_mode <> mode) THEN
					(* Operating mode shanged, returning at the beginning *)
					step				:= 100;
				ELSIF (getSDMstatus.enable = FALSE) AND (getSDMstatus.status = ERR_FUB_ENABLE_FALSE) THEN
					getSDMstatus.enable := TRUE;
					step				:= 11;
				END_IF;

			18:
				(* WRITING ENTRY INTO THE LOGGER *)
				IF (writeLogFlag = TRUE) THEN

					memset(ADR(errorEntry)		,0,	SIZEOF(errorEntry));
					memset(ADR(errorString)		,0,	SIZEOF(errorString));
					memset(ADR(errorStepString)	,0,	SIZEOF(errorStepString));

					errorEntry.errorNum 		:= CST_SDM_ACTIVE;
					errorEntry.logLevel			:= arEVENTLOG_SEVERITY_INFO;
					errorString					:= 'sdmMAN - SDM Active, previous: DISABLED';
					errorEntry.adr_string 		:= ADR(errorString);
					writeError.adrCustomEntry	:= ADR(errorEntry);
					writeError.enable			:= TRUE;
					step 						:= 19;
				ELSE
					step := 19;
				END_IF;
			19:
				(* SDM ACTIVATED  *)
				busy			:= FALSE;
				ready			:= ((writeError.done) AND (writeError.enable)) OR (NOT writeError.enable);
				error			:= FALSE;
				errorID 		:= ERR_OK;
				writeLogFlag 	:= FALSE;
				IF (old_mode <> mode) AND (writeError.done) AND (writeError.enable) THEN
					(* Operating mode shanged, returning at the beginning *)
					step				:= 100;
					writeError.enable	:= FALSE;
				ELSIF (writeError.error AND writeError.enable) THEN
					step := 201;
				ELSIF (old_mode <> mode) AND (NOT writeError.enable) THEN
						(* Operating mode shanged, returning at the beginning *)
						step				:= 100;
						writeError.enable	:= FALSE;
				END_IF;

			20:
				(* If SDM is on the switch it off *)
				IF (old_mode <> mode) THEN
					(* Operating mode shanged, returning at the beginning *)
					step		:= 0;
				ELSIF (getSDMstatus.enable = FALSE) AND (getSDMstatus.status = ERR_FUB_ENABLE_FALSE) THEN
					getSDMstatus.enable := TRUE;
					step		:= 21;
				END_IF;

			21:
				IF (old_mode <> mode) THEN
					(* Operating mode shanged, returning at the beginning *)
					step			:= 100;
				ELSIF (getSDMstatus.status = ERR_OK) AND (getSDMstatus.run = cfgSTATUS_SDM_DISABLED) THEN
					sdmStatus 		:= CST_SDM_DISABLE;
					step			:= 28;
				ELSIF (getSDMstatus.status = ERR_OK) AND (getSDMstatus.run = cfgSTATUS_SDM_ENABLED) THEN
					sdmStatus 		:= CST_SDM_ACTIVE;
					step			:= 22;
					writeLogFlag 	:= TRUE;
				ELSIF (getSDMstatus.status <> ERR_OK) AND (getSDMstatus.status <> ERR_FUB_BUSY) THEN
					(* Error occured *)
					error			:= TRUE;
					errorID			:= getSDMstatus.status;
					errorStep		:= 20;
					step 			:= 200;
				END_IF;

			22:
				(* Disabling the SDM *)
				getSDMstatus.enable		:= FALSE;
				setSDMstatus.enable		:= FALSE;
				IF (old_mode <> mode) THEN
					(* Operating mode shanged, returning at the beginning *)
					step				:= 100;
				ELSIF (getSDMstatus.status = ERR_FUB_ENABLE_FALSE) AND (setSDMstatus.status = ERR_FUB_ENABLE_FALSE) THEN
					setSDMstatus.enable	:= TRUE;
					setSDMstatus.start	:= cfgOPTION_DISABLE_SDM;
					step				:= 23;
				END_IF;

			23:
				IF (old_mode <> mode) THEN
					(* Operating mode shanged, returning at the beginning *)
					step		:= 100;
				ELSIF (setSDMstatus.status = ERR_OK) THEN
					step		:= 24;
				ELSIF (setSDMstatus.status <> ERR_OK) AND (setSDMstatus.status <> ERR_FUB_BUSY) THEN
					(* Error occured *)
					error		:= TRUE;
					errorID		:= setSDMstatus.status;
					errorStep	:= 22;
					step 		:= 200;
				END_IF;

			24:
				(* Reading the sdm status *)
				setSDMstatus.enable	:= FALSE;
				IF (old_mode <> mode) THEN
					(* Operating mode shanged, returning at the beginning *)
					step		:= 100;
				ELSIF (getSDMstatus.enable = FALSE) AND (getSDMstatus.status = ERR_FUB_ENABLE_FALSE) THEN
					getSDMstatus.enable := TRUE;
					step		:= 21;
				END_IF;

			28:
				(* WRITING ENTRY INTO THE LOGGER *)
				IF (writeLogFlag = TRUE) THEN

					memset(ADR(errorEntry)		,0,	SIZEOF(errorEntry));
					memset(ADR(errorString)		,0,	SIZEOF(errorString));
					memset(ADR(errorStepString)	,0,	SIZEOF(errorStepString));

					errorEntry.errorNum 		:= CST_SDM_DISABLE;
					errorEntry.logLevel			:= arEVENTLOG_SEVERITY_INFO;
					errorString					:= 'sdmMAN - SDM DISABLED, previous: ACTIVE';
					errorEntry.adr_string 		:= ADR(errorString);
					writeError.adrCustomEntry	:= ADR(errorEntry);
					writeError.enable			:= TRUE;
					step 						:= 29;
				ELSE
					step := 29;
				END_IF;

			29:
				(* SDM DISABLED *)
				busy	:= FALSE;
				ready	:= ((writeError.done) AND (writeError.enable)) OR (NOT writeError.enable);
				error	:= FALSE;
				errorID := ERR_OK;
				writeLogFlag := FALSE;
				IF (old_mode <> mode) AND (writeError.done) AND (writeError.enable) THEN
					(* Operating mode shanged, returning at the beginning *)
					step				:= 100;
					writeError.enable	:= FALSE;
				ELSIF (writeError.error AND writeError.enable) THEN
					step := 201;
				ELSIF (old_mode <> mode) AND (NOT writeError.enable) THEN
					(* Operating mode shanged, returning at the beginning *)
					step				:= 100;
					writeError.enable	:= FALSE;
				END_IF;

			30:
				(* Manual handling of the sdm configuration *)
				IF (old_mode <> mode) THEN
					(* Operating mode shanged, returning at the beginning *)
					step		:= 0;
				ELSIF (getSDMstatus.enable = FALSE) AND (getSDMstatus.status = ERR_FUB_ENABLE_FALSE) THEN
					getSDMstatus.enable := TRUE;
					step		:= 31;
				END_IF;

			31:
				IF (old_mode <> mode) THEN
					(* Operating mode shanged, returning at the beginning *)
					step		:= 100;
				ELSIF (getSDMstatus.status = ERR_OK) THEN
					sdmStatus 	:= getSDMstatus.run;
					ready 	:= TRUE;
					busy 	:= FALSE;
					error 	:= FALSE;
					IF ((getSDMstatus.run = cfgSTATUS_SDM_DISABLED) AND (reqSDMstatus = cfgOPTION_ENABLE_SDM) OR
						(getSDMstatus.run = cfgSTATUS_SDM_ENABLED) AND (reqSDMstatus = cfgOPTION_DISABLE_SDM)) THEN
						step	:= 32;
					END_IF;

				ELSIF (getSDMstatus.status <> ERR_OK) AND (getSDMstatus.status <> ERR_FUB_BUSY) THEN
					(* Error occured *)
					error		:= TRUE;
					errorID		:= getSDMstatus.status;
					errorStep	:= 30;
					step 		:= 200;
				END_IF;

			32:
				ready 	:= FALSE;
				busy 	:= TRUE;
				error 	:= FALSE;
				(* Changing the SDM configuration *)
				getSDMstatus.enable		:= FALSE;
				setSDMstatus.enable		:= FALSE;
				IF (old_mode <> mode) THEN
					(* Operating mode shanged, returning at the beginning *)
					step				:= 100;
				ELSIF (getSDMstatus.status = ERR_FUB_ENABLE_FALSE) AND (setSDMstatus.status = ERR_FUB_ENABLE_FALSE) THEN
					setSDMstatus.enable	:= TRUE;
					setSDMstatus.start	:= reqSDMstatus;
					step				:= 33;
				END_IF;

			33:
				IF (old_mode <> mode) THEN
					(* Operating mode shanged, returning at the beginning *)
					step		:= 100;
				ELSIF (setSDMstatus.status = ERR_OK) THEN
					step		:= 34;
				ELSIF (setSDMstatus.status <> ERR_OK) AND (setSDMstatus.status <> ERR_FUB_BUSY) THEN
					(* Error occured *)
					error		:= TRUE;
					errorID		:= setSDMstatus.status;
					errorStep	:= 32;
					step 		:= 200;
				END_IF;

			34:
				(* Reading the sdm status *)
				setSDMstatus.enable	:= FALSE;
				IF (old_mode <> mode) THEN
					(* Operating mode shanged, returning at the beginning *)
					step				:= 100;
				ELSIF (getSDMstatus.enable = FALSE) AND (getSDMstatus.status = ERR_FUB_ENABLE_FALSE) THEN
					getSDMstatus.enable	:= TRUE;
					step				:= 35;
				END_IF;

			35:
				IF (getSDMstatus.status = ERR_OK) THEN
					sdmStatus 	:= getSDMstatus.run;
					step	:= 36;
				ELSIF (getSDMstatus.status <> ERR_OK) AND (getSDMstatus.status <> ERR_FUB_BUSY) THEN
				(* Error occured *)
				error		:= TRUE;
				errorID		:= getSDMstatus.status;
				errorStep	:= 34;
				step 		:= 200;
				END_IF;

			36:
				(* WRITING ENTRY INTO THE LOGGER *)
				memset(ADR(errorEntry)		,0,	SIZEOF(errorEntry));
				memset(ADR(errorString)		,0,	SIZEOF(errorString));
				memset(ADR(errorStepString)	,0,	SIZEOF(errorStepString));

				IF (sdmStatus = cfgSTATUS_SDM_DISABLED) THEN
					errorEntry.errorNum 		:= CST_SDM_DISABLE;
					errorString					:= 'sdmMAN - SDM DISABLED, previous: ACTIVE';
				ELSIF (sdmStatus = cfgSTATUS_SDM_ENABLED) THEN
					errorEntry.errorNum 		:= CST_SDM_ACTIVE;
					errorString					:= 'sdmMAN - SDM Active, previous: DISABLED';
				END_IF;

				errorEntry.logLevel			:= arEVENTLOG_SEVERITY_INFO;
				errorEntry.adr_string 		:= ADR(errorString);
				writeError.adrCustomEntry	:= ADR(errorEntry);
				writeError.enable			:= TRUE;
				step 						:= 37;

			37:
				(* SDM DISABLED *)

				IF (writeError.done) AND (writeError.enable) THEN
					(* Operating mode shanged, returning at the beginning *)
					step				:= 31;
					writeError.enable	:= FALSE;
				ELSIF (writeError.error AND writeError.enable) THEN
					step := 201;
					writeError.enable	:= FALSE;
				END_IF;

			40:
				busy 	:= TRUE;
				error	:= FALSE;
				ready	:= FALSE;
				error	:= FALSE;
				errorID	:= FALSE;
				(* SYSTEM DUMP, getting the SDM status *)
				IF (getSDMstatus.status = ERR_FUB_ENABLE_FALSE) THEN
					getSDMstatus.enable := TRUE;
					step := 41;
				END_IF;

			41:
				(* SYSTEM DUMP, getting the SDM status *)
				IF (getSDMstatus.status = ERR_OK) THEN
					sdmStatus		:= getSDMstatus.run;
					oldSdmStatus	:= getSDMstatus.run;
					step			:= 42;
				ELSIF (getSDMstatus.status <> ERR_OK) AND (getSDMstatus.status <> ERR_FUB_BUSY) THEN
				(* Error occured *)
				error		:= TRUE;
				errorID		:= getSDMstatus.status;
				errorStep	:= 40;
				step 		:= 200;
				END_IF;

			42:
				(* SYSTEM DUMP, getting the SDM status *)
				getSDMstatus.enable := FALSE;
				IF (sdmStatus = cfgSTATUS_SDM_DISABLED) AND (getSDMstatus.status = ERR_FUB_ENABLE_FALSE) THEN
					setSDMstatus.start	:= cfgOPTION_ENABLE_SDM;
					setSDMstatus.enable	:= TRUE;
					step			:= 43;
				ELSIF (sdmStatus = cfgSTATUS_SDM_ENABLED) AND (getSDMstatus.status = ERR_FUB_ENABLE_FALSE) THEN
					step			:= 50;
				END_IF;

			43:
				(* SYSTEM DUMP, enabling the SDM *)
				IF (setSDMstatus.status = ERR_OK) THEN
					setSDMstatus.enable := FALSE;
					step				:= 44;
				ELSIF (setSDMstatus.status <> ERR_OK) AND (setSDMstatus.status <> ERR_FUB_BUSY) THEN
					(* Error occured *)
					error		:= TRUE;
					errorID		:= setSDMstatus.status;
					errorStep	:= 42;
					step 		:= 200;
				END_IF;

			44:
				(* SYSTEM DUMP, getting the SDM status *)
				IF (setSDMstatus.status = ERR_FUB_ENABLE_FALSE) THEN
					getSDMstatus.enable := TRUE;
					step := 45;
				END_IF;

			45:
				(* SYSTEM DUMP, getting the SDM status *)
				IF (getSDMstatus.status = ERR_OK) THEN
					sdmStatus 		:= getSDMstatus.run;
					step			:= 46;
				ELSIF (getSDMstatus.status <> ERR_OK) AND (getSDMstatus.status <> ERR_FUB_BUSY) THEN
					(* Error occured *)
					error		:= TRUE;
					errorID		:= getSDMstatus.status;
					errorStep	:= 46;
					step 		:= 200;
				END_IF;

			46:
				(* SYSTEM DUMP, getting the SDM status *)
				getSDMstatus.enable := FALSE;
				IF (getSDMstatus.status = ERR_FUB_ENABLE_FALSE) THEN
					step := 50;
				END_IF;

			50:
				(* SYSTEM DUMP, configuring the DUMP parameters *)
				sDump.configuration := sdm_SYSTEMDUMP_DATA;
				sDump.pFile := 0;
				sDump.pParam := ADR('software,hardware,motion,logger,profiler');
				IF (pDumpDevice <> 0) THEN
					sDump.pDevice := pDumpDevice;
					sDump.enable := TRUE;
					step := 51;
				ELSE
					sDump.enable 	:= FALSE;
					error 			:= TRUE;
					errorStep		:= 50;
					errorID 		:= ERR_BUR_ILLIDENT;
					step := 200;
				END_IF;

			51:
				(* SYSTEM DUMP *)
				IF (pDumpDevice <> sDump.pDevice) THEN
					sDump.enable 	:= FALSE;
					error 			:= TRUE;
					errorStep		:= 50;
					errorID 		:= ERR_BUR_ILLIDENT;
					step := 200;
				ELSIF (sDump.status = ERR_OK) AND (pDumpDevice = sDump.pDevice) THEN
					(* Dump complete, restoring the SDM status *)
					sDump.enable 	:= FALSE;
					step := 60;
				ELSIF (sDump.status <> ERR_OK) AND (sDump.status <> ERR_FUB_BUSY) AND (pDumpDevice = sDump.pDevice) THEN
					sDump.enable 	:= FALSE;
					error 			:= TRUE;
					errorStep		:= 50;
					errorID 		:= sDump.status;
					step := 200;
				END_IF;

			60:
				(* SYSTEM DUMP, reconfiguring the SDM *)
				sDump.enable 	:= FALSE;
				IF (oldSdmStatus <> sdmStatus) THEN
					setSDMstatus.start := oldSdmStatus;
					setSDMstatus.enable	:= TRUE;
					step := 61;
				ELSE
					step := 70;
				END_IF;

			61:
				(* SYSTEM DUMP, reconfiguring the SDM *)
				IF (setSDMstatus.status = ERR_OK) THEN
					setSDMstatus.enable	:= FALSE;
					step := 62;
				ELSIF (setSDMstatus.status <> ERR_OK) AND (setSDMstatus.status <> ERR_FUB_BUSY) THEN
					error 			:= TRUE;
					errorStep		:= 60;
					errorID 		:= setSDMstatus.status;
					step := 200;
				END_IF;

			62:
				(* SYSTEM DUMP, reconfiguring the SDM *)
				IF (setSDMstatus.status = ERR_FUB_ENABLE_FALSE) THEN
					getSDMstatus.enable := TRUE;
					step := 63;
				END_IF;

			63:
				(* SYSTEM DUMP, reconfiguring the SDM *)
				IF (getSDMstatus.status = ERR_OK) THEN
					sdmStatus := getSDMstatus.run;
					getSDMstatus.enable := FALSE;
					step := 60;
				ELSIF (getSDMstatus.status <> ERR_OK) AND (getSDMstatus.status <> ERR_FUB_BUSY) THEN
					error 			:= TRUE;
					errorStep		:= 62;
					errorID 		:= getSDMstatus.status;
					step := 200;
				END_IF;

			70:
				(* SYSTEM DUMP, writing to the logger *)
				memset(ADR(errorEntry)		,0,	SIZEOF(errorEntry));
				memset(ADR(errorString)		,0,	SIZEOF(errorString));
				memset(ADR(errorStepString)	,0,	SIZEOF(errorStepString));

				errorEntry.errorNum 		:= CST_SDM_DUMP_DONE;
				errorEntry.logLevel			:= arEVENTLOG_SEVERITY_INFO;
				errorString					:= 'sdmMAN - System Dump Created';
				errorEntry.adr_string 		:= ADR(errorString);
				writeError.adrCustomEntry	:= ADR(errorEntry);
				writeError.enable			:= TRUE;
				step 						:= 71;

			71:
			(* SYSTEM DUMP, writing to the logger *)
				IF writeError.done THEN
					writeError.enable 	:= FALSE;
					step 				:= 79;
				ELSIF	writeError.error THEN
					writeError.enable 	:= FALSE;
					internalError 		:= TRUE;
					step 				:= 202;
				END_IF;

			79:
				(* SYSTEM DUMP, completed *)
				busy := FALSE;
				ready := TRUE;
				error := FALSE;
				errorID := ERR_OK;
				IF (old_mode <> mode) THEN
					(* Operating mode shanged, returning at the beginning *)
					step				:= 100;
				END_IF;

			100:
				(* Disabling used function blocks *)
				getSDMstatus.enable := FALSE;
				setSDMstatus.enable	:= FALSE;
				IF (getSDMstatus.status = ERR_FUB_ENABLE_FALSE) AND (setSDMstatus.status = ERR_FUB_ENABLE_FALSE) THEN
					step := 0;
				END_IF;

			200:
				(* Error state, disabling all the used function  blocks and writing the error into the logger *)
				getSDMstatus.enable			:= FALSE;
				setSDMstatus.enable			:= FALSE;

				memset(ADR(errorEntry)		,0,	SIZEOF(errorEntry));
				memset(ADR(errorString)		,0,	SIZEOF(errorString));
				memset(ADR(errorStepString)	,0,	SIZEOF(errorStepString));

				errorEntry.errorNum 		:= errorID;
				errorEntry.logLevel			:= arEVENTLOG_SEVERITY_WARNING;
				errorString					:= 'sdmMAN - Error step: ';
				itoa(USINT_TO_DINT(errorStep),	ADR(errorStepString));
				strcat(ADR(errorString)		, 	ADR(errorStepString));
				errorEntry.adr_string 		:= ADR(errorString);
				writeError.adrCustomEntry	:= ADR(errorEntry);
				writeError.enable			:= TRUE;
				step 						:= 201;

			201:
				getSDMstatus.enable			:= FALSE;
				setSDMstatus.enable			:= FALSE;

				IF writeError.done THEN
					writeError.enable 	:= FALSE;
					step 				:= 202;
				ELSIF	writeError.error THEN
					writeError.enable 	:= FALSE;
					internalError 		:= TRUE;
					step 				:= 202;
				END_IF;

			202:
				(* Waiting to disable the function block *)

		END_CASE;

	ELSE

		(* Function block disabled *)
		busy				:= FALSE;
		ready				:= FALSE;
		error				:= TRUE;
		errorID				:= ERR_FUB_ENABLE_FALSE;
		internalError 		:= FALSE;
		writeLogFlag 		:= FALSE;
		errorStep			:= 0;
		step				:= 0;
		sdmStatus			:= 0;
		oldSdmStatus		:= 0;
		(* Disabling used function blocks *)
		getSDMstatus.enable	:= FALSE;
		setSDMstatus.enable	:= FALSE;
		writeError.enable	:= FALSE;
		sDump.enable		:= FALSE;

	END_IF;

	getSDMstatus();
	setSDMstatus();
	writeError();
	sDump();
END_FUNCTION_BLOCK

(* ---- SearchIO.st ---- *)
(********************************************************************
 * COPYRIGHT -- Microsoft
 ********************************************************************
 * Library: Powertoys
 * File: SearchIO.st
 * Author: Paolino
 * Created: April 18, 2014
 ********************************************************************
 * Implementation of library Powertoys
 ********************************************************************)

(* Function Block to show hardware list component *)
FUNCTION_BLOCK SearchIO

	IF (enable	=	TRUE) THEN

		CASE step OF

			0:
				(* Getting the information from configured and/or inserted hardware modules  *)

				FB_DiagCreateInfo.enable	:=	TRUE;
				FB_DiagCreateInfo.infoKind	:=	mode;

				errorID 		:=	ERR_FUB_BUSY;
				busy			:=	TRUE;
				error			:=	FALSE;

				IF (FB_DiagCreateInfo.status	=	ERR_FUB_BUSY) THEN
					(* The function block started running *)
					step :=	1;
				END_IF;

			1:
				IF (FB_DiagCreateInfo.status	=	ERR_OK) THEN

					(* Collecting data *)
					ident	     			:=	FB_DiagCreateInfo.ident;
					nrEntries	 			:=	FB_DiagCreateInfo.nrEntries;

					(* Disabling the used fub *)
					FB_DiagCreateInfo.enable 	:=	FALSE;

					IF (wholeList = TRUE) THEN
						(* Create the whole hw list *)
						step        				:=	10;
					ELSE
						(* Output only the specified index *)
						step						:=	60;
					END_IF;

				ELSIF ((FB_DiagCreateInfo.status	<>	ERR_OK)	AND	(FB_DiagCreateInfo.status	<>	ERR_FUB_BUSY)) THEN
					(* Going to the error state *)
					errorID		:=	FB_DiagCreateInfo.status;
					errorStep	:=	1;
					step		:=	200;
					error		:=	TRUE;
				END_IF

			10:
				(* Getting path of inserted hardware modules *)
				pData ACCESS (adrSearchIO + (SIZEOF (pData))*counter);
				IF (counter <= (nrEntries - 1)) THEN
					FB_DiagGetStrInfo.infoCode		:=	asdiagPATH;
					FB_DiagGetStrInfo.index			:=	counter;
					FB_DiagGetStrInfo.ident			:=	ident;
					FB_DiagGetStrInfo.pBuffer		:=	ADR(pData.Path);
					FB_DiagGetStrInfo.bufferLen		:=	SIZEOF (pData.Path) - 1;
					FB_DiagGetStrInfo.enable		:=	TRUE;

					//IF (FB_DiagGetStrInfo.status	=	ERR_FUB_BUSY) THEN
						step := 11;
					//END_IF

				ELSE

					counter						:=	0;
					FB_DiagGetStrInfo.enable 	:=	FALSE;
					step 						:= 	13;

				END_IF

			11:
				IF (FB_DiagGetStrInfo.status	=	ERR_OK) THEN

					counter						:=	counter + 1;
					FB_DiagGetStrInfo.enable 	:=	FALSE;
					step 						:=	12;

				ELSIF (FB_DiagGetStrInfo.status	<>	ERR_FUB_BUSY)	AND	(FB_DiagGetStrInfo.status	<>	ERR_OK) THEN
					(* Going to the error state *)
					errorID		:=	FB_DiagGetStrInfo.status;
					errorStep	:=	10;
					step		:=	200;
					error		:=	TRUE;

				END_IF

			12:

				IF (FB_DiagGetStrInfo.status	=	ERR_FUB_ENABLE_FALSE) THEN

					step	:=	10;
				END_IF

			13:
				IF (FB_DiagGetStrInfo.status	=	ERR_FUB_ENABLE_FALSE) THEN

					step	:=	20;

				END_IF

			20:
				(*Getting Model Number of inserted hardware modules*)
				pData ACCESS (adrSearchIO + SIZEOF (pData)*counter);
				IF (counter <= (nrEntries -1)) THEN
					FB_DiagGetStrInfo.infoCode	:=	asdiagPLUGGED_MODULE;
					FB_DiagGetStrInfo.index		:=	counter;
					FB_DiagGetStrInfo.ident		:=	ident;
					FB_DiagGetStrInfo.pBuffer	:=	ADR(pData.ModelNumber);
					FB_DiagGetStrInfo.bufferLen	:=	SIZEOF(pData.ModelNumber) - 1;
					FB_DiagGetStrInfo.enable	:=	TRUE;

					//IF (FB_DiagGetStrInfo.status	=	ERR_FUB_BUSY) THEN
						step := 21;
					//END_IF

				ELSE

					counter						:=	0;
					FB_DiagGetStrInfo.enable 	:=	FALSE;
					step 						:= 	23;

				END_IF

			21:
				IF (FB_DiagGetStrInfo.status	=	ERR_OK) THEN

					counter						:=	counter + 1;
					FB_DiagGetStrInfo.enable 	:=	FALSE;
					step 						:=	22;

				ELSIF (FB_DiagGetStrInfo.status	<>	ERR_FUB_BUSY)	AND	(FB_DiagGetStrInfo.status	<>	ERR_OK) THEN
					(* Going to the error state *)
					errorID		:=	FB_DiagGetStrInfo.status;
					errorStep	:=	20;
					step		:=	200;
					error		:=	TRUE;

				END_IF

			22:

				IF (FB_DiagGetStrInfo.status	=	ERR_FUB_ENABLE_FALSE) THEN

					step	:=	20;
				END_IF

			23:
				IF (FB_DiagGetStrInfo.status	=	ERR_FUB_ENABLE_FALSE) THEN

					step	:=	30;

				END_IF

			30:
				(*Getting Name of inserted hardware modules*)
				pData ACCESS (adrSearchIO + SIZEOF (pData)*counter);
				IF (counter <= (nrEntries -1)) THEN
					FB_DiagGetStrInfo.infoCode	:=	asdiagHARDWARE_MODULE_NAME;
					FB_DiagGetStrInfo.index		:=	counter;
					FB_DiagGetStrInfo.ident		:=	ident;
					FB_DiagGetStrInfo.pBuffer	:=	ADR(pData.Name);
					FB_DiagGetStrInfo.bufferLen	:=	SIZEOF(pData.Name) - 1;
					FB_DiagGetStrInfo.enable	:=	TRUE;

					//IF (FB_DiagGetStrInfo.status	=	ERR_FUB_BUSY) THEN
						step := 31;
					//END_IF

				ELSE

					counter				:=	0;
					FB_DiagGetStrInfo.enable 	:=	FALSE;
					step 						:= 	33;

				END_IF

			31:
				IF (FB_DiagGetStrInfo.status	=	ERR_OK) THEN

					counter						:=	counter + 1;
					FB_DiagGetStrInfo.enable 	:=	FALSE;
					step 						:=	32;

				ELSIF (FB_DiagGetStrInfo.status	<>	ERR_FUB_BUSY)	AND	(FB_DiagGetStrInfo.status	<>	ERR_OK) THEN
					(* Going to the error state *)
					errorID		:=	FB_DiagGetStrInfo.status;
					errorStep	:=	30;
					step		:=	200;
					error		:=	TRUE;

				END_IF

			32:

				IF (FB_DiagGetStrInfo.status	=	ERR_FUB_ENABLE_FALSE) THEN

					step	:=	30;
				END_IF

			33:
				IF (FB_DiagGetStrInfo.status	=	ERR_FUB_ENABLE_FALSE) THEN

					step	:=	50;

				END_IF

			50:
				(*Getting Serial Number of hardware modules*)
				pData ACCESS (adrSearchIO + SIZEOF (pData)*counter);
				IF (counter <= (nrEntries -1)) THEN
					FB_DiagGetNumInfo.ident		:=	ident;
					FB_DiagGetNumInfo.index		:=	counter;
					FB_DiagGetNumInfo.infoCode	:=	asdiagSERIAL_NUMBER;
					FB_DiagGetNumInfo.enable	:=	TRUE;

					//IF (FB_DiagGetNumInfo.status = ERR_FUB_BUSY) THEN
						step := 51;
					//END_IF

				ELSE

					counter						:=	0;
					FB_DiagGetNumInfo.enable	:=	FALSE;
					step						:=	53;

				END_IF

			51:
				IF (FB_DiagGetNumInfo.status	=	ERR_OK) THEN

					pData.Serial 					:=	FB_DiagGetNumInfo.value;
					counter							:=	counter +1;
					FB_DiagGetNumInfo.enable		:=	FALSE;
					step := 52;

				ELSIF (FB_DiagGetNumInfo.status	<>	ERR_FUB_BUSY)	AND	(FB_DiagGetNumInfo.status	<>	ERR_OK) THEN
					(* Going to the error state *)
					errorID		:=	FB_DiagGetNumInfo.status;
					errorStep	:=	50;
					step		:=	200;
					error		:=	TRUE;

				END_IF

			52:

				IF (FB_DiagGetNumInfo.status	=	ERR_FUB_ENABLE_FALSE) THEN

					step	:=	50;
				END_IF

			53:
				IF (FB_DiagGetNumInfo.status	=	ERR_FUB_ENABLE_FALSE) THEN

					step	:=	100;

				END_IF
			(**************************************************************************************)
			(***************** Output only the specified stationIndex *****************************)
			(**************************************************************************************)
			60:
				(* Getting path of specified hw module *)
				pData ACCESS (adrSearchIO);
				FB_DiagGetStrInfo.infoCode		:=	asdiagPATH;
				FB_DiagGetStrInfo.index			:=	stationIndex;
				FB_DiagGetStrInfo.ident			:=	ident;
				FB_DiagGetStrInfo.pBuffer		:=	ADR(pData.Path);
				FB_DiagGetStrInfo.bufferLen		:=	SIZEOF (pData.Path) - 1;
				FB_DiagGetStrInfo.enable		:=	TRUE;

				step := 61;

			61:
				IF (FB_DiagGetStrInfo.status	=	ERR_OK) THEN

					FB_DiagGetStrInfo.enable 	:=	FALSE;
					step 						:=	62;

				ELSIF (FB_DiagGetStrInfo.status	<>	ERR_FUB_BUSY)	AND	(FB_DiagGetStrInfo.status	<>	ERR_OK) THEN
					(* Going to the error state *)
					errorID		:=	FB_DiagGetStrInfo.status;
					errorStep	:=	60;
					step		:=	200;
					error		:=	TRUE;

				END_IF

			62:
				IF (FB_DiagGetStrInfo.status	=	ERR_FUB_ENABLE_FALSE) THEN

					step	:=	63;

				END_IF

			63:
				(*Getting Model Number of inserted hardware modules*)
				FB_DiagGetStrInfo.infoCode	:=	asdiagPLUGGED_MODULE;
				FB_DiagGetStrInfo.index		:=	stationIndex;
				FB_DiagGetStrInfo.ident		:=	ident;
				FB_DiagGetStrInfo.pBuffer	:=	ADR(pData.ModelNumber);
				FB_DiagGetStrInfo.bufferLen	:=	SIZEOF(pData.ModelNumber) - 1;
				FB_DiagGetStrInfo.enable	:=	TRUE;

				step := 64;

			64:
				IF (FB_DiagGetStrInfo.status	=	ERR_OK) THEN

					FB_DiagGetStrInfo.enable 	:=	FALSE;
					step 						:=	65;

				ELSIF (FB_DiagGetStrInfo.status	<>	ERR_FUB_BUSY)	AND	(FB_DiagGetStrInfo.status	<>	ERR_OK) THEN
					(* Going to the error state *)
					errorID		:=	FB_DiagGetStrInfo.status;
					errorStep	:=	63;
					step		:=	200;
					error		:=	TRUE;

				END_IF

			65:

				IF (FB_DiagGetStrInfo.status	=	ERR_FUB_ENABLE_FALSE) THEN

					step	:=	66;
				END_IF

			66:
				(*Getting Name of inserted hardware modules*)

				FB_DiagGetStrInfo.infoCode	:=	asdiagHARDWARE_MODULE_NAME;
				FB_DiagGetStrInfo.index		:=	stationIndex;
				FB_DiagGetStrInfo.ident		:=	ident;
				FB_DiagGetStrInfo.pBuffer	:=	ADR(pData.Name);
				FB_DiagGetStrInfo.bufferLen	:=	SIZEOF(pData.Name) - 1;
				FB_DiagGetStrInfo.enable	:=	TRUE;

				step := 67;

			67:
				IF (FB_DiagGetStrInfo.status	=	ERR_OK) THEN

					FB_DiagGetStrInfo.enable 	:=	FALSE;
					step 						:=	68;

				ELSIF (FB_DiagGetStrInfo.status	<>	ERR_FUB_BUSY)	AND	(FB_DiagGetStrInfo.status	<>	ERR_OK) THEN
					(* Going to the error state *)
					errorID		:=	FB_DiagGetStrInfo.status;
					errorStep	:=	66;
					step		:=	200;
					error		:=	TRUE;

				END_IF

			68:
				IF (FB_DiagGetStrInfo.status	=	ERR_FUB_ENABLE_FALSE) THEN

					step	:=	69;

				END_IF

			69:
				(*Getting Serial Number of hardware modules*)
				FB_DiagGetNumInfo.ident		:=	ident;
				FB_DiagGetNumInfo.index		:=	stationIndex;
				FB_DiagGetNumInfo.infoCode	:=	asdiagSERIAL_NUMBER;
				FB_DiagGetNumInfo.enable	:=	TRUE;

				step := 70;

			70:
				IF (FB_DiagGetNumInfo.status	=	ERR_OK) THEN

					pData.Serial 					:=	FB_DiagGetNumInfo.value;
					FB_DiagGetNumInfo.enable		:=	FALSE;
					step := 71;

				ELSIF (FB_DiagGetNumInfo.status	<>	ERR_FUB_BUSY)	AND	(FB_DiagGetNumInfo.status	<>	ERR_OK) THEN
					(* Going to the error state *)
					errorID		:=	FB_DiagGetNumInfo.status;
					errorStep	:=	69;
					step		:=	200;
					error		:=	TRUE;

				END_IF

			71:
				IF (FB_DiagGetNumInfo.status	=	ERR_FUB_ENABLE_FALSE) THEN

					step	:=	100;

				END_IF

			100:
				done 			:= TRUE;
				busy 			:= FALSE;
				errorID 		:= ERR_OK;

				FB_DiagCreateInfo.enable		:= FALSE;
				FB_DiagGetStrInfo.enable		:= FALSE;
				FB_DiagGetNumInfo.enable		:= FALSE;

			200:
				(* Error step *)
//				FB_DiagCreateInfo.enable		:= FALSE;
//				FB_DiagGetStrInfo.enable		:= FALSE;
//				FB_DiagGetNumInfo.enable		:= FALSE;

				done				:= TRUE;
				busy				:= FALSE;
				error 				:= TRUE;

		END_CASE;

	ELSE
		(* Function block not enabled *)
		error				:= TRUE;
		errorID				:= ERR_FUB_ENABLE_FALSE;

		(* Resetting  the internal variables *)
		errorStep			:= 0;
		step	 			:= 0;
		ident 				:= 0;
		counter 			:= 0;
		nrEntries 			:= 0;

		done				:= FALSE;
		busy				:= FALSE;

		(* Disabling the block *)
		FB_DiagCreateInfo.enable		:= FALSE;
		FB_DiagGetStrInfo.enable		:= FALSE;
		FB_DiagGetNumInfo.enable		:= FALSE;

	END_IF;

	(*Function Block Call*)
	FB_DiagCreateInfo();
	FB_DiagGetStrInfo();
	FB_DiagGetNumInfo();

END_FUNCTION_BLOCK

(* ---- Powertoys.var ---- *)
(********************************************************************
 * COPYRIGHT -- Bernecker + Rainer
 ********************************************************************
 * Library: Powertoys
 * File: Powertoys.var
 * Author: gibertinim
 * Created: March 27, 2014
 ********************************************************************
 * Constants of library Powertoys
 ********************************************************************)
VAR CONSTANT
	CST_SW_OBJ_CHANGED : UINT := 55100; (*Software object changed*)
	CST_SDM_DISABLE : UINT := 55110; (*Disable SDM*)
	CST_SDM_ACTIVE : UINT := 55111; (*Activate SDM*)
	CST_SDM_DUMP_DONE : UINT := 55112; (*System dump completed*)
	CST_NO_NTC : UINT := 55120; (*No network command trace available*)
END_VAR
